INTERFACE I_Strategy

METHOD execute
VAR_INPUT
	in_rDistance		:REAL;
END_VAR
END_METHOD

END_INTERFACE

(* stored: Version 1.1.0.1
   Itf I_Strategy: Id {695c9049-7b34-46b0-ae5a-a740e04831f2}
   Method execute: Id {bf14d6c7-87cd-4a33-a26b-5e6304addf78} *)
